ABB RAPID module: TCP_moratool2.mod

MODULE TCP_moratool2
	! Points are read in order of declaration.
  ! Please do not change the order of points!

  LOCAL PERS robtarget pTCP_Point1:=[[740.698,82.7345,312.832],[0.135539,0.133535,-0.9796,-0.0646607],[0,0,-1,0],[9E+9,9E+9,9E+9,9E+9,9E+9,9E+9]];
	LOCAL PERS robtarget pTCP_Point2:=[[470.306,64.9459,200.532],[0.85501,0.0108509,0.516619,0.0441084],[0,0,0,1],[9E+9,9E+9,9E+9,9E+9,9E+9,9E+9]];
	LOCAL PERS robtarget pTCP_Point3:=[[611.169,239.139,215.826],[0.221167,-0.168067,0.721243,-0.634545],[0,0,2,1],[9E+9,9E+9,9E+9,9E+9,9E+9,9E+9]];
	LOCAL PERS robtarget pTCP_Point4:=[[602.267,-92.8862,210.336],[0.69256,-0.626606,0.164581,0.317235],[-1,0,1,0],[9E+9,9E+9,9E+9,9E+9,9E+9,9E+9]];

ENDMODULE
